# EPICS substitutions: ipimbLib/Db/archive_ipimb.substitutions
#
# ipimb archive substitutions file
#

# Generate ipimb archive file
#	Macros:
#		TODO:	List here any macros used in the template
#				Note which ones have defaults.
file archive_ipimb.template
{
	{
		# Hack till msi supports empty substitutions
		IOC		=	$(IOC),
	}
}
